// TIA Portal project "project_box_stacking" (V18)
// Vorlageprojekt für das Buch mit Zielsystem S7-1200

(* hardware
DEVICE "S7-1200-Station_1"  S7-1200 Station
   slot 0: "Baugruppenträger_0"  Rack  V1.0
   slot 1: "PLC_1"  CPU 1211C DC/DC/DC  6ES7 211-1AE40-0XB0  V4.1
*)

// ===== PLC "PLC_1"  CPU 1211C DC/DC/DC =====

VAR_GLOBAL   // PLC tag table "Standard-Variablentabelle"
   "FirstScan" AT %M1.0 : Bool;
   "DiagStatusUpdate" AT %M1.1 : Bool;
   "AlwaysTRUE" AT %M1.2 : Bool;
   "AlwaysFALSE" AT %M1.3 : Bool;
   "Clock_Byte" AT %MB0 : Byte;
   "Clock_10Hz" AT %M0.0 : Bool;
   "Clock_5Hz" AT %M0.1 : Bool;
   "Clock_2.5Hz" AT %M0.2 : Bool;
   "Clock_2Hz" AT %M0.3 : Bool;
   "Clock_1.25Hz" AT %M0.4 : Bool;
   "Clock_1Hz" AT %M0.5 : Bool;
   "Clock_0.625Hz" AT %M0.6 : Bool;
   "Clock_0.5Hz" AT %M0.7 : Bool;
   "System_Byte" AT %MB1 : Byte;
END_VAR

VAR_GLOBAL   // PLC tag table " FactoryIO_1"
   "Moving X" AT %I0.0 : Bool;
   "Moving Z" AT %I0.1 : Bool;
   "Item detected" AT %I0.2 : Bool;
   "Lid before place" AT %I0.3 : Bool;
   "Lid clamped" AT %I0.4 : Bool;
   "Pos. at limit (lids)" AT %I0.5 : Bool;
   "Base at place" AT %I0.6 : Bool;
   "Base clamped" AT %I0.7 : Bool;
   "Pos. at limit (bases)" AT %I1.0 : Bool;
   "Part leaving" AT %I1.1 : Bool;
   "Start" AT %I1.2 : Bool;
   "Reset" AT %I1.3 : Bool;
   "Stop" AT %I1.4 : Bool;
   "Emergency stop" AT %I1.5 : Bool;
   "Auto" AT %I1.6 : Bool;
   "FACTORY I/O (Running)" AT %I1.7 : Bool;
   "Grab" AT %Q0.2 : Bool;
   "Lids conveyor" AT %Q0.3 : Bool;
   "Clamp lid" AT %Q0.4 : Bool;
   "Pos. raise (lids)" AT %Q0.5 : Bool;
   "Bases conveyor" AT %Q0.6 : Bool;
   "Pos. raise (bases)" AT %Q1.0 : Bool;
   "Start light" AT %Q1.1 : Bool;
   "Reset light" AT %Q1.2 : Bool;
   "Stop light" AT %Q1.3 : Bool;
   "Counter" AT %QD31 : DInt;
   "Clamp base" AT %Q0.7 : Bool;
   "Move X" AT %Q0.0 : Bool;
   "Move Z" AT %Q0.1 : Bool;
   "Vision sensor Blue lid" AT %I2.4 : Bool;
   "Green Light" AT %Q1.4 : Bool;
   "Counter stacked" AT %I2.3 : Bool;
   "Lid queue" AT %I2.2 : Bool;
   "Sensor stacked" AT %I2.1 : Bool;
   "FACTORY I/O (Reset)" AT %I2.0 : Bool;
   "Vision sensor Blue base" AT %I2.5 : Bool;
   "sensor lid at place" AT %I2.6 : Bool;
   "Base leaving" AT %I2.7 : Bool;
   "Sensor bases at place" AT %I5.3 : Bool;
END_VAR

VAR_GLOBAL   // PLC tag table " FactoryIO_2"
   "Moving X 2" AT %I3.0 : Bool;
   "Moving Z 2" AT %I3.1 : Bool;
   "Item detected 2" AT %I3.2 : Bool;
   "Lid before place 2" AT %I3.3 : Bool;
   "Lid clamped 2" AT %I3.4 : Bool;
   "Pos. at limit (lids) 2" AT %I3.5 : Bool;
   "Base at place 2" AT %I3.6 : Bool;
   "Base clamped 2" AT %I3.7 : Bool;
   "Pos. at limit (bases) 2" AT %I4.0 : Bool;
   "Part leaving 2" AT %I4.1 : Bool;
   "Sensor stacked 2" AT %I4.2 : Bool;
   "Lid queue 2" AT %I4.3 : Bool;
   "Counter stacked 2" AT %I4.4 : Bool;
   "Vision Sensor Green Lid" AT %I4.5 : Bool;
   "Move X 2" AT %Q2.0 : Bool;
   "Move Z 2" AT %Q2.1 : Bool;
   "Grab 2" AT %Q2.2 : Bool;
   "Lids conveyor 2" AT %Q2.3 : Bool;
   "Clamp lid 2" AT %Q2.4 : Bool;
   "Pos. raise (lids) 2" AT %Q2.5 : Bool;
   "Counter 2" AT %QD35 : DInt;
   "Bases conveyor 2" AT %Q2.6 : Bool;
   "Clamp base 2" AT %Q2.7 : Bool;
   "Pos. raise (bases) 2" AT %Q3.0 : Bool;
   "Sensor lid at place 2" AT %I4.6 : Bool;
   "Vision Sensor Green Base" AT %I4.7 : Bool;
   "Base leaving 2" AT %I5.0 : Bool;
   "Sensor base at place 2" AT %I5.1 : Bool;
END_VAR

VAR_GLOBAL   // PLC tag table "markers"
   "m_is_system_on" AT %M3.0 : Bool;
   "m_lid_conveyor" AT %M3.1 : Bool;
   "m_base_conveyor" AT %M3.2 : Bool;
END_VAR

DATA_BLOCK "FB_main_DB"   // DB1
{ S7_Optimized_Access := 'TRUE' }
VERSION : 0.1
// stored: InstanceOfName FB_main
"FB_main"
BEGIN
END_DATA_BLOCK

DATA_BLOCK "FB_main_DB_2"   // DB2
{ S7_Optimized_Access := 'TRUE' }
VERSION : 0.1
// stored: InstanceOfName FB_main
"FB_main"
BEGIN
END_DATA_BLOCK

FUNCTION_BLOCK "FB_main"   // FB1, LAD
{ S7_Optimized_Access := 'TRUE' }
VERSION : 0.1
   VAR_INPUT
      iReset : Bool;   // 'Reset button status' - Observes the reset button, used to reset the system to initial conditions
      iLid_before_place : Bool;   // iLid_at_place - 'Lid presence sensor' - Detects whether a lid is at the required position to be fit
      iItem_detected : Bool;   // 'Item detection sensor' - Identifies the presence of an item in a robotic arm
      iBase_before_place : Bool;   // 'Base presence sensor' - Senses if a base is present at the required position to be fit
      iPart_leaving : Bool;   // Part departure sensor' - Monitors parts leaving a grip area, to control the flow of items.
      iSensor_stacked : Bool;   // 'Stack sensor' - Detects stacked items
      iLid_clamped : Bool;   // - Checks the lid mechanism is clamped,
      iBase_clamped : Bool;   // Checks the basesmechanism is clamped,
      iMoving_Z : Bool;   // Detects movement along the Z-axis,
      iMoving_X : Bool;   // Detects movement along the X-axis
      iLid_queue : Bool;   // Monitors the place before lids grab area
      iCounter_stacked : Bool;   // Stack counter' - Counts the number of stacked items
      iVision_sensor_blue_lid : Bool;   // Blue lid vision sensor' - Vision system input that detects the presence of blue-colored lids;
      iVision_sensor_blue_base : Bool;   // Blue lid vision sensor' - Vision system input that detects the presence of blue-colored lids;
      "iSensor_lid _at_place" : Bool;   // Checks for the presence of a lid at the pick-up point.
      "iSensor_base _at_place" : Bool;   // Checks for the presence of a base at the pick-up point.
      iBase_leaving : Bool;   // "Monitors for a objects leaving pick up point
   END_VAR
   VAR_OUTPUT
      "qLid_ conveyor" : Bool;   // 'Conveyor belt control for lid transport' - Activates the conveyor section responsible for moving lids/parts
      "qBase_ conveyor" : Bool;   // 'Conveyor belt control for base transport' - Activates the conveyor section for moving the base parts
      qClamp_lid : Bool;   // 'Actuate lid clamp' - Engages the mechanism to clamp the lid
      qClamp_base : Bool;   // 'Actuate base clamp' - Engages the mechanism to clamp the base
      qMove_Z : Bool;   // 'Vertical movement actuator' - Controls the vertical movement, likely of a robotic arm
      qMove_X : Bool;   // 'Horizontal movement actuator X-axis' - Controls the horizontal movement along the X-axis
      qGrab : Bool;   // 'Gripping actuator control' - Activates the mechanism to grip an item
      "qPos._raise_lids" : Bool;   // 'Conveyor lids passage control mechanism' - Controls the raising and lowering mechanism
      "qPos._raise_bases" : Bool;   // 'Conveyor bases passage control mechanism' - Controls the raising and lowering mechanism
      qCount_stacked : DInt;   // 'Stack count monitoring' - display the count of stacked items at exit
      qGreen_light : Bool;   // 'Green light indicator' - Activates the green light
   END_VAR
   VAR
      Sequence_lids : Struct
         is_at_place : Bool;
         is_fited : Bool;
         is_grabed : Bool;
         is_above_base : Bool;
      END_STRUCT;
      Sequence_bases : Struct
         at_place : Bool := false;
         is_fited : Bool := false;
      END_STRUCT;
      Sequence_part : Struct
         is_stacked : Bool;
         above_lids_conv : Bool;
         at_place : Bool;
         "exit" : Bool;
      END_STRUCT;
      sequence_no_blue : Struct
         lids : Bool;
         bases : Bool;
      END_STRUCT;
      "array" : Array[0..10] of Bool;
      onemove : Bool;   // System flag to make one operation in program
      Timer_1 : TON_TIME;
      Timer_2 : TON_TIME;
      Timer_3 : TON_TIME;
      Timer_4 : TON_TIME;
      Timer_5 : TON_TIME;
      Timer_6 : TON_TIME;
      Timer_7 : TON_TIME;
      Timer_8 : TON_TIME;
      Timer_9 : TON_TIME;
      Timer_10 : TON_TIME;
      Timer_11 : TON_TIME;
      Timer_12 : TON_TIME;
      "counter" : CTU_INT;   // "stacked parts counter at exit - Tracks the number of completed cycles or parts processed.
   END_VAR
   VAR RETAIN
      reset : Bool;   // System Reset Flag
   END_VAR
   VAR_TEMP   // added for the SCL form of the ladder/FBD networks
      _w1 : Bool;
      _w2 : Bool;
      _w3 : Bool;
   END_VAR
BEGIN

REGION Network 1: init
   // Initialization Routine - Resets control bits and status indicators at system startup or upon reset. Ensures that the system begins operation with a clear configuration
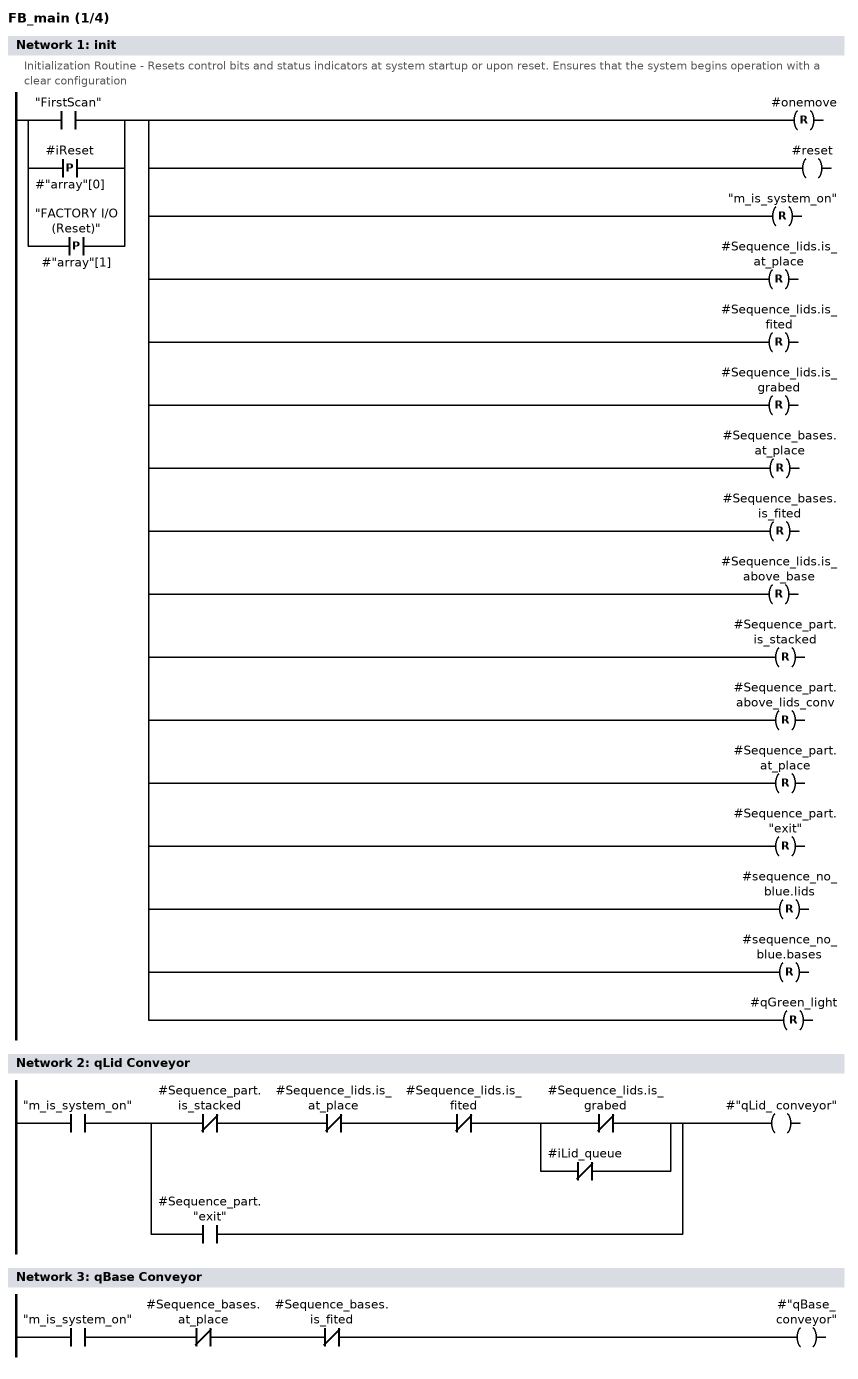
   RUNG wire#powerrail
      Contact( "FirstScan" )
      wire#w1
      R_Coil( #onemove )
   END_RUNG
   RUNG wire#powerrail
      P_Contact(operand := #iReset, bit := #"array"[0])
   END_RUNG wire#w1
   RUNG wire#powerrail
      P_Contact(operand := "FACTORY I/O (Reset)", bit := #"array"[1])
   END_RUNG wire#w1
   RUNG wire#w1
      Coil( #reset )
   END_RUNG
   RUNG wire#w1
      R_Coil( "m_is_system_on" )
   END_RUNG
   RUNG wire#w1
      R_Coil( #Sequence_lids.is_at_place )
   END_RUNG
   RUNG wire#w1
      R_Coil( #Sequence_lids.is_fited )
   END_RUNG
   RUNG wire#w1
      R_Coil( #Sequence_lids.is_grabed )
   END_RUNG
   RUNG wire#w1
      R_Coil( #Sequence_bases.at_place )
   END_RUNG
   RUNG wire#w1
      R_Coil( #Sequence_bases.is_fited )
   END_RUNG
   RUNG wire#w1
      R_Coil( #Sequence_lids.is_above_base )
   END_RUNG
   RUNG wire#w1
      R_Coil( #Sequence_part.is_stacked )
   END_RUNG
   RUNG wire#w1
      R_Coil( #Sequence_part.above_lids_conv )
   END_RUNG
   RUNG wire#w1
      R_Coil( #Sequence_part.at_place )
   END_RUNG
   RUNG wire#w1
      R_Coil( #Sequence_part."exit" )
   END_RUNG
   RUNG wire#w1
      R_Coil( #sequence_no_blue.lids )
   END_RUNG
   RUNG wire#w1
      R_Coil( #sequence_no_blue.bases )
   END_RUNG
   RUNG wire#w1
      R_Coil( #qGreen_light )
   END_RUNG
   // the same network as SCL:
   #_w1 := #iReset AND NOT #"array"[0];   // rising edge of #iReset
   #"array"[0] := #iReset;
   #_w2 := "FACTORY I/O (Reset)" AND NOT #"array"[1];   // rising edge of "FACTORY I/O (Reset)"
   #"array"[1] := "FACTORY I/O (Reset)";
   #_w3 := "FirstScan" OR #_w1 OR #_w2;
   IF #_w3 THEN #onemove := FALSE; END_IF;
   #reset := #_w3;
   IF #_w3 THEN
       "m_is_system_on" := FALSE;
       #Sequence_lids.is_at_place := FALSE;
       #Sequence_lids.is_fited := FALSE;
       #Sequence_lids.is_grabed := FALSE;
       #Sequence_bases.at_place := FALSE;
       #Sequence_bases.is_fited := FALSE;
       #Sequence_lids.is_above_base := FALSE;
       #Sequence_part.is_stacked := FALSE;
       #Sequence_part.above_lids_conv := FALSE;
       #Sequence_part.at_place := FALSE;
       #Sequence_part."exit" := FALSE;
       #sequence_no_blue.lids := FALSE;
       #sequence_no_blue.bases := FALSE;
       #qGreen_light := FALSE;
   END_IF;
END_REGION

REGION Network 2: qLid Conveyor
   RUNG wire#powerrail
      Contact( "m_is_system_on" )
      wire#w1
      I_Contact( #Sequence_part.is_stacked )
      I_Contact( #Sequence_lids.is_at_place )
      I_Contact( #Sequence_lids.is_fited )
      wire#w2
      I_Contact( #Sequence_lids.is_grabed )
      wire#w3
      Coil( #"qLid_ conveyor" )
   END_RUNG
   RUNG wire#w2
      I_Contact( #iLid_queue )
   END_RUNG wire#w3
   RUNG wire#w1
      Contact( #Sequence_part."exit" )
   END_RUNG wire#w3
   // the same network as SCL:
   #"qLid_ conveyor" := "m_is_system_on" AND ((NOT #Sequence_part.is_stacked AND NOT #Sequence_lids.is_at_place AND NOT #Sequence_lids.is_fited AND (NOT #Sequence_lids.is_grabed OR NOT #iLid_queue)) OR #Sequence_part."exit");
END_REGION

REGION Network 3: qBase Conveyor
   RUNG wire#powerrail
      Contact( "m_is_system_on" )
      I_Contact( #Sequence_bases.at_place )
      I_Contact( #Sequence_bases.is_fited )
      Coil( #"qBase_ conveyor" )
   END_RUNG
   // the same network as SCL:
   #"qBase_ conveyor" := "m_is_system_on" AND NOT #Sequence_bases.at_place AND NOT #Sequence_bases.is_fited;
END_REGION

REGION Network 4: qClamp lid
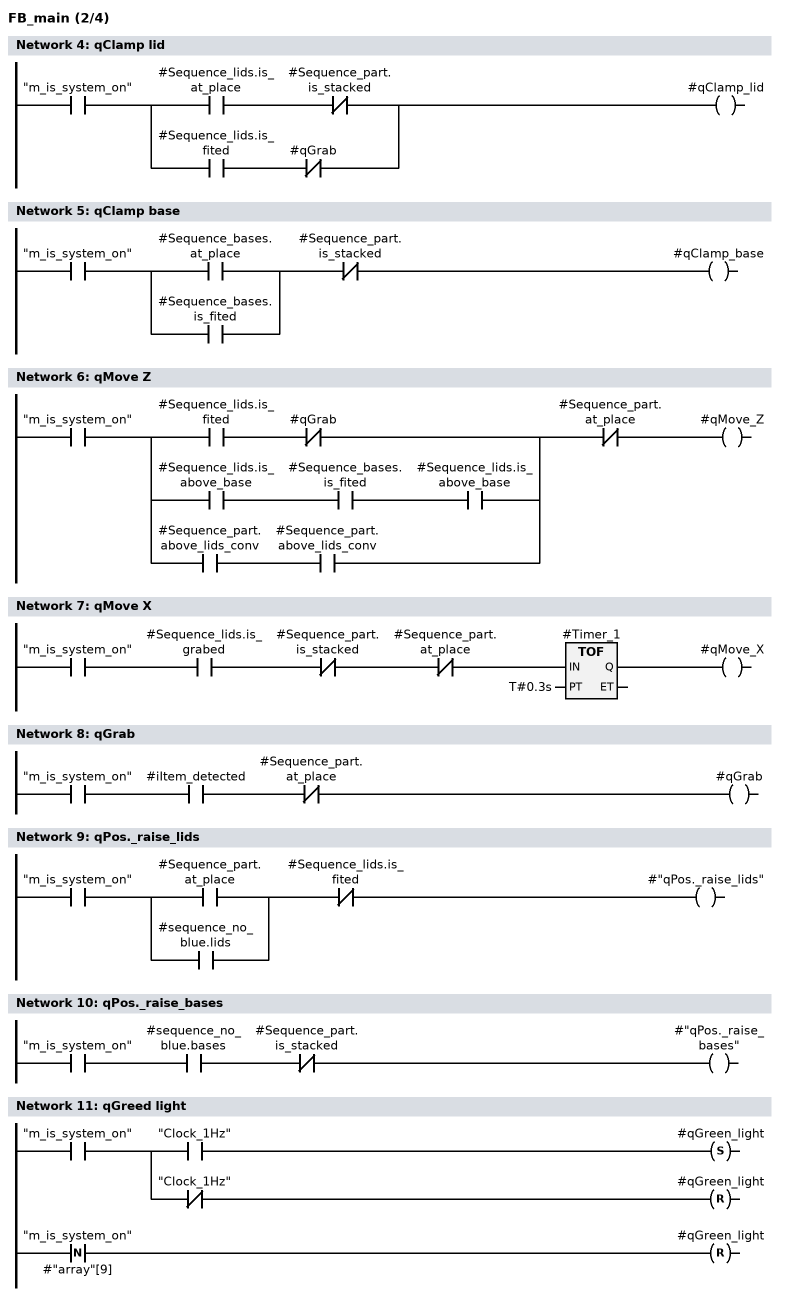
   RUNG wire#powerrail
      Contact( "m_is_system_on" )
      wire#w1
      Contact( #Sequence_lids.is_at_place )
      I_Contact( #Sequence_part.is_stacked )
      wire#w2
      Coil( #qClamp_lid )
   END_RUNG
   RUNG wire#w1
      Contact( #Sequence_lids.is_fited )
      I_Contact( #qGrab )
   END_RUNG wire#w2
   // the same network as SCL:
   #qClamp_lid := "m_is_system_on" AND ((#Sequence_lids.is_at_place AND NOT #Sequence_part.is_stacked) OR (#Sequence_lids.is_fited AND NOT #qGrab));
END_REGION

REGION Network 5: qClamp base
   RUNG wire#powerrail
      Contact( "m_is_system_on" )
      wire#w1
      Contact( #Sequence_bases.at_place )
      wire#w2
      I_Contact( #Sequence_part.is_stacked )
      Coil( #qClamp_base )
   END_RUNG
   RUNG wire#w1
      Contact( #Sequence_bases.is_fited )
   END_RUNG wire#w2
   // the same network as SCL:
   #qClamp_base := "m_is_system_on" AND (#Sequence_bases.at_place OR #Sequence_bases.is_fited) AND NOT #Sequence_part.is_stacked;
END_REGION

REGION Network 6: qMove Z
   RUNG wire#powerrail
      Contact( "m_is_system_on" )
      wire#w1
      Contact( #Sequence_lids.is_fited )
      I_Contact( #qGrab )
      wire#w2
      I_Contact( #Sequence_part.at_place )
      Coil( #qMove_Z )
   END_RUNG
   RUNG wire#w1
      Contact( #Sequence_lids.is_above_base )
      Contact( #Sequence_bases.is_fited )
      Contact( #Sequence_lids.is_above_base )
   END_RUNG wire#w2
   RUNG wire#w1
      Contact( #Sequence_part.above_lids_conv )
      Contact( #Sequence_part.above_lids_conv )
   END_RUNG wire#w2
   // the same network as SCL:
   #qMove_Z := "m_is_system_on" AND ((#Sequence_lids.is_fited AND NOT #qGrab) OR (#Sequence_lids.is_above_base AND #Sequence_bases.is_fited AND #Sequence_lids.is_above_base) OR (#Sequence_part.above_lids_conv AND #Sequence_part.above_lids_conv)) AND NOT #Sequence_part.at_place;
END_REGION

REGION Network 7: qMove X
   #Timer_1(IN := "m_is_system_on" AND #Sequence_lids.is_grabed AND NOT #Sequence_part.is_stacked AND NOT #Sequence_part.at_place,   // TOF
            PT := T#0.3s);
   #qMove_X := #Timer_1.Q;
END_REGION

REGION Network 8: qGrab
   RUNG wire#powerrail
      Contact( "m_is_system_on" )
      Contact( #iItem_detected )
      I_Contact( #Sequence_part.at_place )
      Coil( #qGrab )
   END_RUNG
   // the same network as SCL:
   #qGrab := "m_is_system_on" AND #iItem_detected AND NOT #Sequence_part.at_place;
END_REGION

REGION Network 9: qPos._raise_lids
   RUNG wire#powerrail
      Contact( "m_is_system_on" )
      wire#w1
      Contact( #Sequence_part.at_place )
      wire#w2
      I_Contact( #Sequence_lids.is_fited )
      Coil( #"qPos._raise_lids" )
   END_RUNG
   RUNG wire#w1
      Contact( #sequence_no_blue.lids )
   END_RUNG wire#w2
   // the same network as SCL:
   #"qPos._raise_lids" := "m_is_system_on" AND (#Sequence_part.at_place OR #sequence_no_blue.lids) AND NOT #Sequence_lids.is_fited;
END_REGION

REGION Network 10: qPos._raise_bases
   RUNG wire#powerrail
      Contact( "m_is_system_on" )
      Contact( #sequence_no_blue.bases )
      I_Contact( #Sequence_part.is_stacked )
      Coil( #"qPos._raise_bases" )
   END_RUNG
   // the same network as SCL:
   #"qPos._raise_bases" := "m_is_system_on" AND #sequence_no_blue.bases AND NOT #Sequence_part.is_stacked;
END_REGION

REGION Network 11: qGreed light
   RUNG wire#powerrail
      Contact( "m_is_system_on" )
      wire#w1
      Contact( "Clock_1Hz" )
      S_Coil( #qGreen_light )
   END_RUNG
   RUNG wire#w1
      I_Contact( "Clock_1Hz" )
      R_Coil( #qGreen_light )
   END_RUNG
   RUNG wire#powerrail
      N_Contact(operand := "m_is_system_on", bit := #"array"[9])
      R_Coil( #qGreen_light )
   END_RUNG
   // the same network as SCL:
   IF "m_is_system_on" AND "Clock_1Hz" THEN #qGreen_light := TRUE; END_IF;
   IF "m_is_system_on" AND NOT "Clock_1Hz" THEN #qGreen_light := FALSE; END_IF;
   #_w1 := NOT "m_is_system_on" AND #"array"[9];   // falling edge of "m_is_system_on"
   #"array"[9] := "m_is_system_on";
   IF #_w1 THEN #qGreen_light := FALSE; END_IF;
END_REGION

REGION Network 12: Sequence lids at place
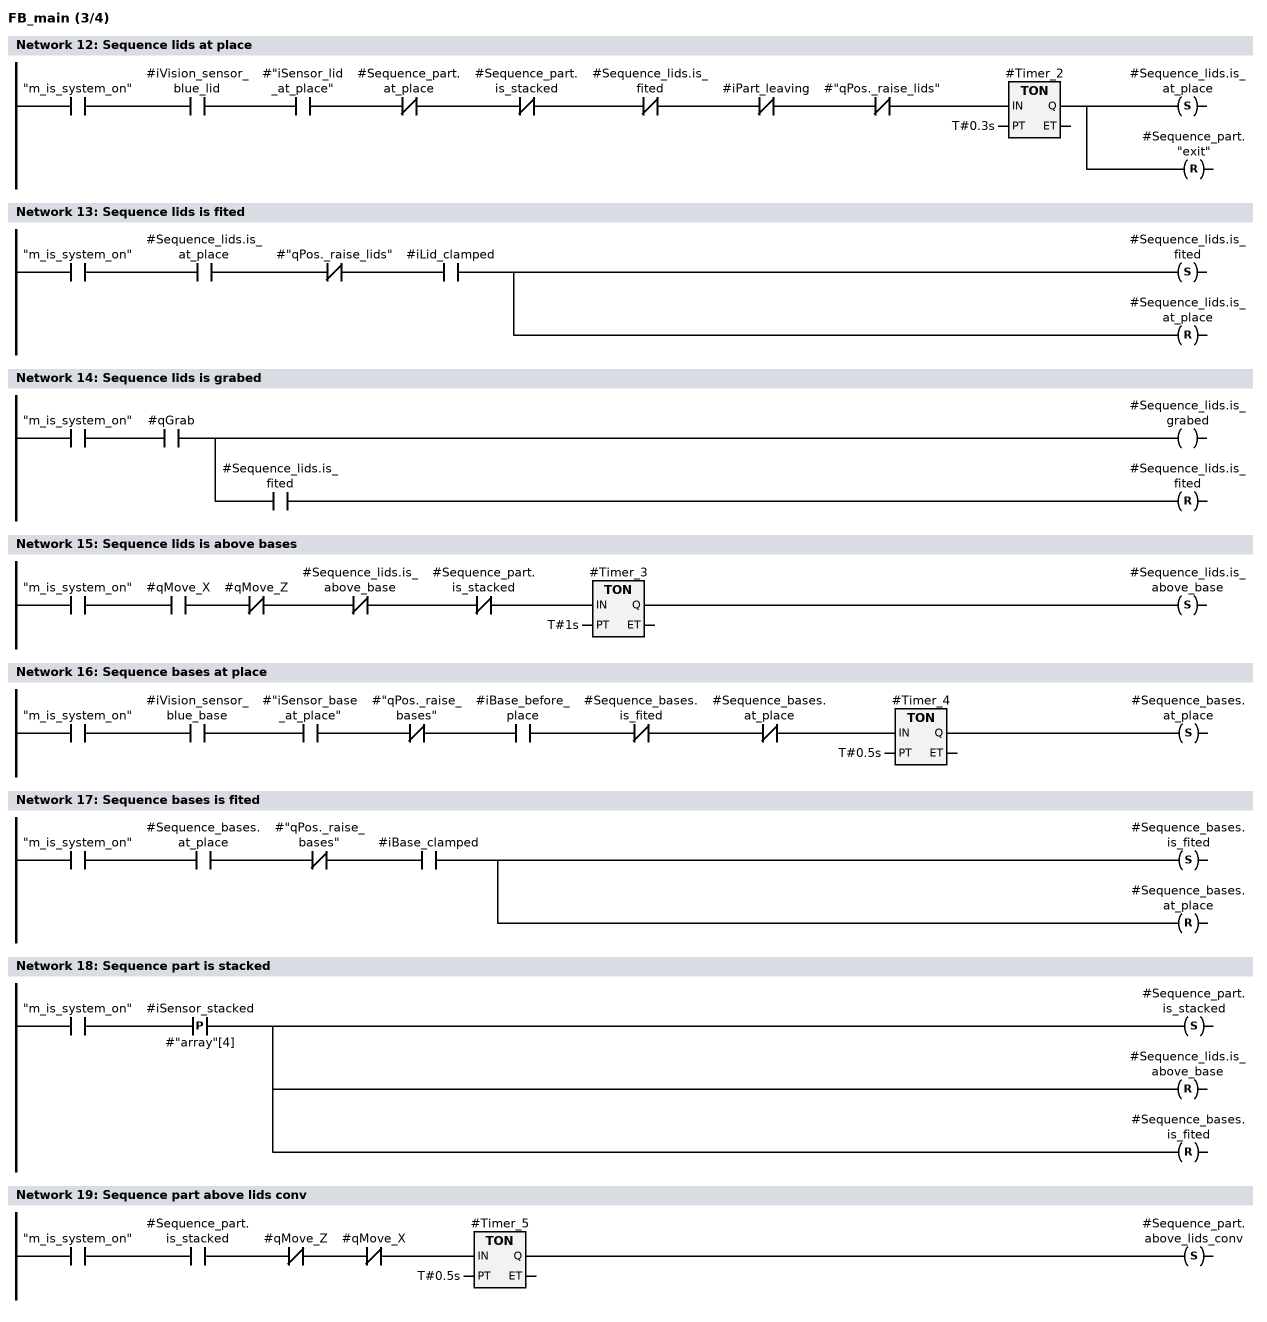
   #Timer_2(IN := "m_is_system_on" AND #iVision_sensor_blue_lid AND #"iSensor_lid _at_place" AND NOT #Sequence_part.at_place AND NOT #Sequence_part.is_stacked AND NOT #Sequence_lids.is_fited AND NOT #iPart_leaving AND NOT #"qPos._raise_lids",   // TON
            PT := T#0.3s);
   IF #Timer_2.Q THEN
       #Sequence_lids.is_at_place := TRUE;
       #Sequence_part."exit" := FALSE;
   END_IF;
END_REGION

REGION Network 13: Sequence lids is fited
   RUNG wire#powerrail
      Contact( "m_is_system_on" )
      Contact( #Sequence_lids.is_at_place )
      I_Contact( #"qPos._raise_lids" )
      Contact( #iLid_clamped )
      wire#w1
      S_Coil( #Sequence_lids.is_fited )
   END_RUNG
   RUNG wire#w1
      R_Coil( #Sequence_lids.is_at_place )
   END_RUNG
   // the same network as SCL:
   IF "m_is_system_on" AND #Sequence_lids.is_at_place AND NOT #"qPos._raise_lids" AND #iLid_clamped THEN
       #Sequence_lids.is_fited := TRUE;
       #Sequence_lids.is_at_place := FALSE;
   END_IF;
END_REGION

REGION Network 14: Sequence lids is grabed
   RUNG wire#powerrail
      Contact( "m_is_system_on" )
      Contact( #qGrab )
      wire#w1
      Coil( #Sequence_lids.is_grabed )
   END_RUNG
   RUNG wire#w1
      Contact( #Sequence_lids.is_fited )
      R_Coil( #Sequence_lids.is_fited )
   END_RUNG
   // the same network as SCL:
   #Sequence_lids.is_grabed := "m_is_system_on" AND #qGrab;
   IF #Sequence_lids.is_grabed AND #Sequence_lids.is_fited THEN #Sequence_lids.is_fited := FALSE; END_IF;
END_REGION

REGION Network 15: Sequence lids is above bases
   #Timer_3(IN := "m_is_system_on" AND #qMove_X AND NOT #qMove_Z AND NOT #Sequence_lids.is_above_base AND NOT #Sequence_part.is_stacked,   // TON
            PT := T#1s);
   IF #Timer_3.Q THEN #Sequence_lids.is_above_base := TRUE; END_IF;
END_REGION

REGION Network 16: Sequence bases at place
   #Timer_4(IN := "m_is_system_on" AND #iVision_sensor_blue_base AND #"iSensor_base _at_place" AND NOT #"qPos._raise_bases" AND #iBase_before_place AND NOT #Sequence_bases.is_fited AND NOT #Sequence_bases.at_place,   // TON
            PT := T#0.5s);
   IF #Timer_4.Q THEN #Sequence_bases.at_place := TRUE; END_IF;
END_REGION

REGION Network 17: Sequence bases is fited
   RUNG wire#powerrail
      Contact( "m_is_system_on" )
      Contact( #Sequence_bases.at_place )
      I_Contact( #"qPos._raise_bases" )
      Contact( #iBase_clamped )
      wire#w1
      S_Coil( #Sequence_bases.is_fited )
   END_RUNG
   RUNG wire#w1
      R_Coil( #Sequence_bases.at_place )
   END_RUNG
   // the same network as SCL:
   IF "m_is_system_on" AND #Sequence_bases.at_place AND NOT #"qPos._raise_bases" AND #iBase_clamped THEN
       #Sequence_bases.is_fited := TRUE;
       #Sequence_bases.at_place := FALSE;
   END_IF;
END_REGION

REGION Network 18: Sequence part is stacked
   RUNG wire#powerrail
      Contact( "m_is_system_on" )
      P_Contact(operand := #iSensor_stacked, bit := #"array"[4])
      wire#w1
      S_Coil( #Sequence_part.is_stacked )
   END_RUNG
   RUNG wire#w1
      R_Coil( #Sequence_lids.is_above_base )
   END_RUNG
   RUNG wire#w1
      R_Coil( #Sequence_bases.is_fited )
   END_RUNG
   // the same network as SCL:
   #_w1 := "m_is_system_on" AND #iSensor_stacked AND NOT #"array"[4];   // rising edge of #iSensor_stacked
   #"array"[4] := #iSensor_stacked;
   IF #_w1 THEN
       #Sequence_part.is_stacked := TRUE;
       #Sequence_lids.is_above_base := FALSE;
       #Sequence_bases.is_fited := FALSE;
   END_IF;
END_REGION

REGION Network 19: Sequence part above lids conv
   #Timer_5(IN := "m_is_system_on" AND #Sequence_part.is_stacked AND NOT #qMove_Z AND NOT #qMove_X,   // TON
            PT := T#0.5s);
   IF #Timer_5.Q THEN #Sequence_part.above_lids_conv := TRUE; END_IF;
END_REGION

REGION Network 20: Sequence part at place
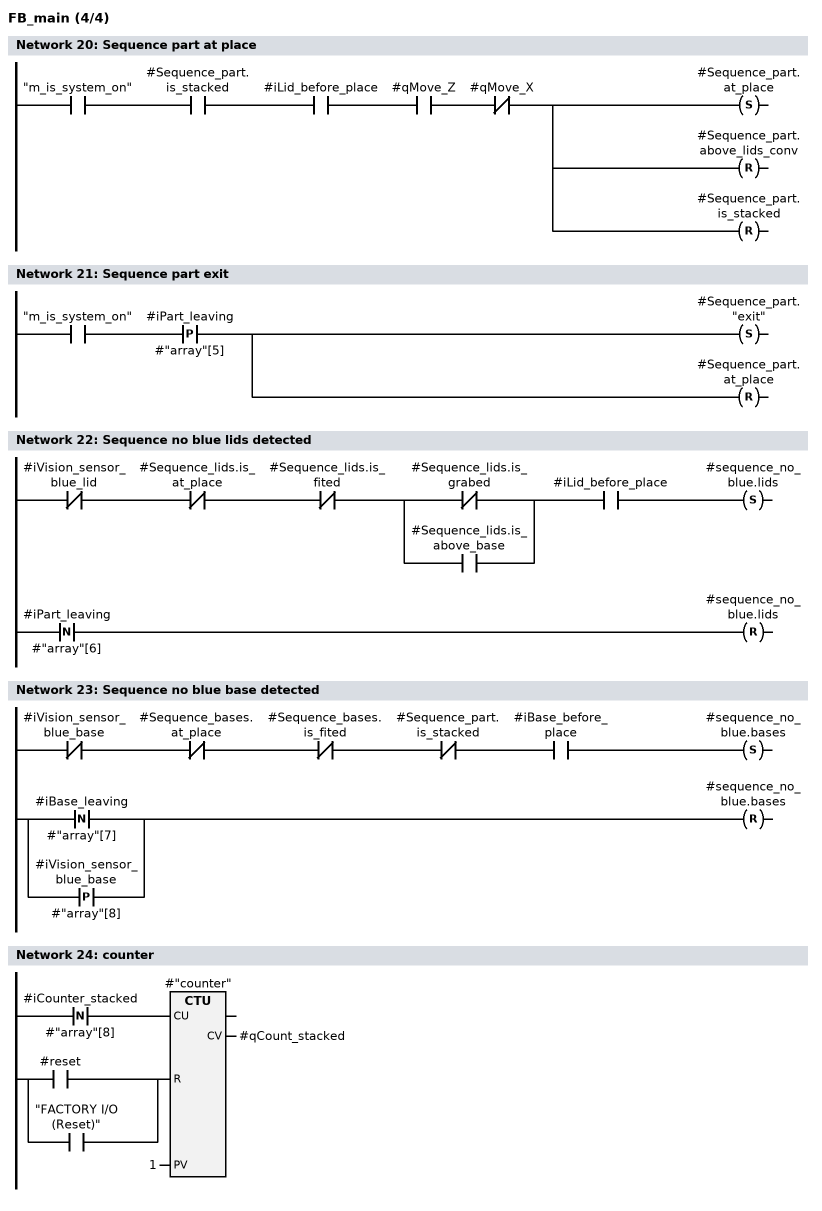
   RUNG wire#powerrail
      Contact( "m_is_system_on" )
      Contact( #Sequence_part.is_stacked )
      Contact( #iLid_before_place )
      Contact( #qMove_Z )
      I_Contact( #qMove_X )
      wire#w1
      S_Coil( #Sequence_part.at_place )
   END_RUNG
   RUNG wire#w1
      R_Coil( #Sequence_part.above_lids_conv )
   END_RUNG
   RUNG wire#w1
      R_Coil( #Sequence_part.is_stacked )
   END_RUNG
   // the same network as SCL:
   IF "m_is_system_on" AND #Sequence_part.is_stacked AND #iLid_before_place AND #qMove_Z AND NOT #qMove_X THEN
       #Sequence_part.at_place := TRUE;
       #Sequence_part.above_lids_conv := FALSE;
       #Sequence_part.is_stacked := FALSE;
   END_IF;
END_REGION

REGION Network 21: Sequence part exit
   RUNG wire#powerrail
      Contact( "m_is_system_on" )
      P_Contact(operand := #iPart_leaving, bit := #"array"[5])
      wire#w1
      S_Coil( #Sequence_part."exit" )
   END_RUNG
   RUNG wire#w1
      R_Coil( #Sequence_part.at_place )
   END_RUNG
   // the same network as SCL:
   #_w1 := "m_is_system_on" AND #iPart_leaving AND NOT #"array"[5];   // rising edge of #iPart_leaving
   #"array"[5] := #iPart_leaving;
   IF #_w1 THEN
       #Sequence_part."exit" := TRUE;
       #Sequence_part.at_place := FALSE;
   END_IF;
END_REGION

REGION Network 22: Sequence no blue lids detected
   RUNG wire#powerrail
      I_Contact( #iVision_sensor_blue_lid )
      I_Contact( #Sequence_lids.is_at_place )
      I_Contact( #Sequence_lids.is_fited )
      wire#w1
      I_Contact( #Sequence_lids.is_grabed )
      wire#w2
      Contact( #iLid_before_place )
      S_Coil( #sequence_no_blue.lids )
   END_RUNG
   RUNG wire#w1
      Contact( #Sequence_lids.is_above_base )
   END_RUNG wire#w2
   RUNG wire#powerrail
      N_Contact(operand := #iPart_leaving, bit := #"array"[6])
      R_Coil( #sequence_no_blue.lids )
   END_RUNG
   // the same network as SCL:
   IF NOT #iVision_sensor_blue_lid AND NOT #Sequence_lids.is_at_place AND NOT #Sequence_lids.is_fited AND (NOT #Sequence_lids.is_grabed OR #Sequence_lids.is_above_base) AND #iLid_before_place THEN
       #sequence_no_blue.lids := TRUE;
   END_IF;
   #_w1 := NOT #iPart_leaving AND #"array"[6];   // falling edge of #iPart_leaving
   #"array"[6] := #iPart_leaving;
   IF #_w1 THEN #sequence_no_blue.lids := FALSE; END_IF;
END_REGION

REGION Network 23: Sequence no blue base detected
   RUNG wire#powerrail
      I_Contact( #iVision_sensor_blue_base )
      I_Contact( #Sequence_bases.at_place )
      I_Contact( #Sequence_bases.is_fited )
      I_Contact( #Sequence_part.is_stacked )
      Contact( #iBase_before_place )
      S_Coil( #sequence_no_blue.bases )
   END_RUNG
   RUNG wire#powerrail
      N_Contact(operand := #iBase_leaving, bit := #"array"[7])
      wire#w1
      R_Coil( #sequence_no_blue.bases )
   END_RUNG
   RUNG wire#powerrail
      P_Contact(operand := #iVision_sensor_blue_base, bit := #"array"[8])
   END_RUNG wire#w1
   // the same network as SCL:
   IF NOT #iVision_sensor_blue_base AND NOT #Sequence_bases.at_place AND NOT #Sequence_bases.is_fited AND NOT #Sequence_part.is_stacked AND #iBase_before_place THEN
       #sequence_no_blue.bases := TRUE;
   END_IF;
   #_w1 := NOT #iBase_leaving AND #"array"[7];   // falling edge of #iBase_leaving
   #"array"[7] := #iBase_leaving;
   #_w2 := #iVision_sensor_blue_base AND NOT #"array"[8];   // rising edge of #iVision_sensor_blue_base
   #"array"[8] := #iVision_sensor_blue_base;
   IF #_w1 OR #_w2 THEN #sequence_no_blue.bases := FALSE; END_IF;
END_REGION

REGION Network 24: counter
   #_w1 := NOT #iCounter_stacked AND #"array"[8];   // falling edge of #iCounter_stacked
   #"array"[8] := #iCounter_stacked;
   #"counter"(CU := #_w1, R := #reset OR "FACTORY I/O (Reset)", PV := 1, CV => #qCount_stacked);   // CTU
END_REGION

REGION Network 25: need to base conveyor
END_REGION
END_FUNCTION_BLOCK

FUNCTION "system on/off" : Void   // FC1, LAD
{ S7_Optimized_Access := 'TRUE' }
VERSION : 0.1
   VAR_INPUT
      iStart_button : Bool;
      iStop_button : Bool;
   END_VAR
BEGIN

REGION Network 1
   // System Control Logic - Monitors the start and stop conditions to maintain the system's operational state. Ensures that the system can only be started if it is not signaled to stop or reset.
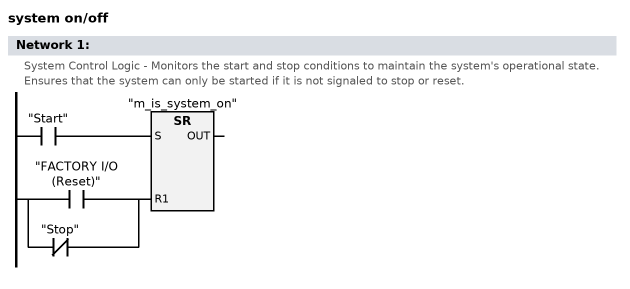
   RUNG wire#powerrail
      Contact( "Start" )
      S_SR(operand := "m_is_system_on", r1 := wire#w1)
   END_RUNG
   RUNG wire#powerrail
      Contact( "FACTORY I/O (Reset)" )
   END_RUNG wire#w1
   RUNG wire#powerrail
      I_Contact( "Stop" )
   END_RUNG wire#w1
   // the same network as SCL:
   IF "Start" THEN
       "m_is_system_on" := TRUE;   // SR flip-flop
   END_IF;
   IF "FACTORY I/O (Reset)" OR NOT "Stop" THEN "m_is_system_on" := FALSE; END_IF;
END_REGION
END_FUNCTION

FUNCTION "MHJ-PLC-Lab-Function-S71200" : Void   // FC9000, SCL
{ S7_Optimized_Access := 'TRUE' }
VERSION : 0.1
   VAR_TEMP
      rdTimeReturn : Int;
      outputTime : DTL;
      SyncVal : Byte;
      forVal : Int;
      forVal_2 : Int;
      Value : Byte;
   END_VAR
   VAR CONSTANT
      CompVal : Byte := 16#34;
      Value_01 : Byte := 16#11;
      Value_01_DW : DWord := 16#A165_D992;
      Value_02_DW : DWord := 16#58BE_4401;
   END_VAR
BEGIN

   #Value:=PEEK(area := 16#82,
        dbNumber := 0,
        byteOffset := 511);
   #Value := #Value + 1;

   POKE(area := 16#82,
        dbNumber := 0,
        byteOffset := 511,
        value := #Value);

   POKE(area:=16#81,
        dbNumber:=0,
        byteOffset:=1016,
        value:=#Value_01_DW);
   POKE(area := 16#81,
        dbNumber := 0,
        byteOffset := 1020,
        value := #Value_02_DW);

   POKE(area := 16#81,
        dbNumber := 0,
        byteOffset := 511,
        value := B#16#00);

   FOR #forVal := 0 TO 120 DO
       FOR #forVal_2:=0 TO 10 DO
           #rdTimeReturn:=RD_SYS_T(#outputTime);
           #rdTimeReturn := WR_SYS_T(#outputTime);
           #rdTimeReturn := RD_SYS_T(#outputTime);
           #rdTimeReturn := WR_SYS_T(#outputTime);
       END_FOR;
       #SyncVal:= PEEK(area := 16#81,
                      dbNumber := 0,
                      byteOffset := 511);
       IF #SyncVal = #CompVal THEN
          GOTO M_1;
       END_IF;
   END_FOR;
   RETURN;

   M_1:
   POKE(area := 16#81,
        dbNumber := 0,
        byteOffset := 511,
        value := B#16#0);
END_FUNCTION

ORGANIZATION_BLOCK "Main"   // OB1, LAD, ProgramCycle
TITLE = "Main Program Sweep (Cycle)"
{ S7_Optimized_Access := 'TRUE' }
VERSION : 0.1
   VAR_INPUT
      Initial_Call : Bool;   // Initial call of this OB
      Remanence : Bool;   // =True, if remanent data are available
   END_VAR
BEGIN

REGION Network 1: Konnektierungsbaustein für PLC-Lab
   // Im Netzwerk 1 wird der Konnektierungsbaustein für PLC-Lab aufgerufen.
   // Dieser Aufruf darf nicht entfernt werden!
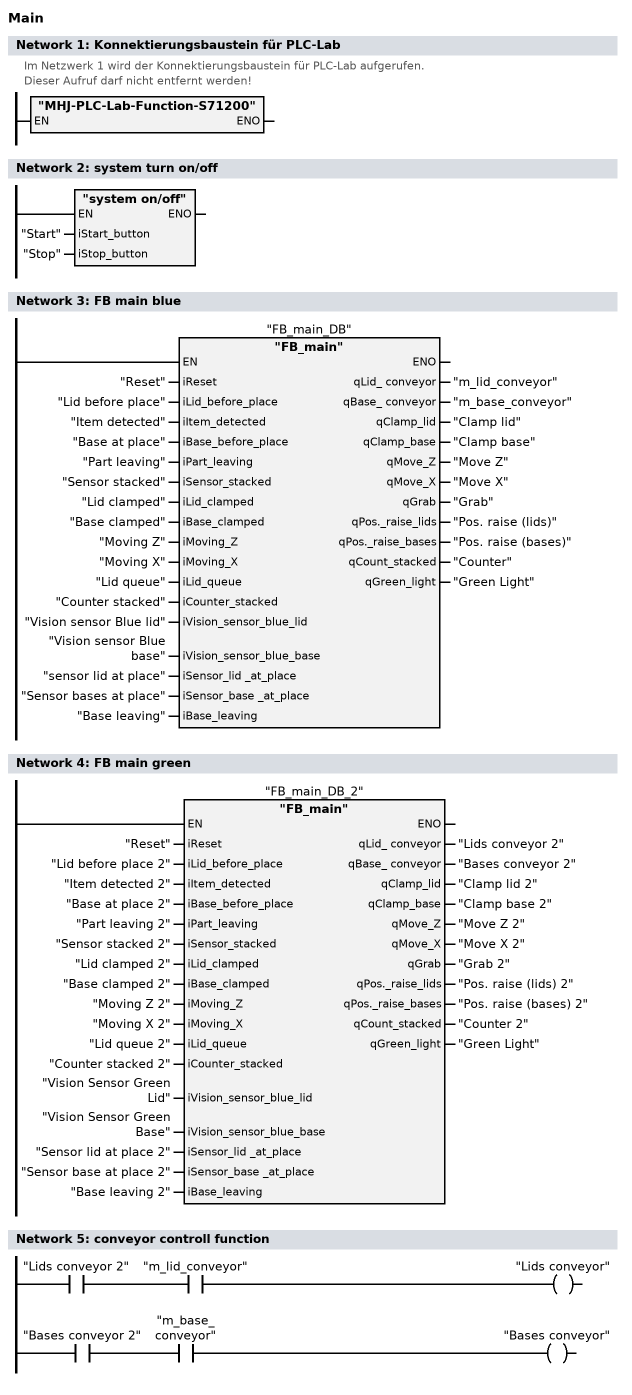
   RUNG wire#powerrail
      "MHJ-PLC-Lab-Function-S71200"()
   END_RUNG
   // the same network as SCL:
   "MHJ-PLC-Lab-Function-S71200"();
END_REGION

REGION Network 2: system turn on/off
   RUNG wire#powerrail
      "system on/off"(iStart_button := "Start", iStop_button := "Stop")
   END_RUNG
   // the same network as SCL:
   "system on/off"(iStart_button := "Start", iStop_button := "Stop");
END_REGION

REGION Network 3: FB main blue
   RUNG wire#powerrail
      "FB_main_DB"(iReset := "Reset", iLid_before_place := "Lid before place", iItem_detected := "Item detected", iBase_before_place := "Base at place", iPart_leaving := "Part leaving", iSensor_stacked := "Sensor stacked", iLid_clamped := "Lid clamped", iBase_clamped := "Base clamped", iMoving_Z := "Moving Z", iMoving_X := "Moving X", iLid_queue := "Lid queue", iCounter_stacked := "Counter stacked", iVision_sensor_blue_lid := "Vision sensor Blue lid", iVision_sensor_blue_base := "Vision sensor Blue base", "iSensor_lid _at_place" := "sensor lid at place", "iSensor_base _at_place" := "Sensor bases at place", iBase_leaving := "Base leaving", "qLid_ conveyor" => "m_lid_conveyor", "qBase_ conveyor" => "m_base_conveyor", qClamp_lid => "Clamp lid", qClamp_base => "Clamp base", qMove_Z => "Move Z", qMove_X => "Move X", qGrab => "Grab", "qPos._raise_lids" => "Pos. raise (lids)", "qPos._raise_bases" => "Pos. raise (bases)", qCount_stacked => "Counter", qGreen_light => "Green Light")
   END_RUNG
   // the same network as SCL:
   "FB_main_DB"(iReset := "Reset",   // "FB_main"
                iLid_before_place := "Lid before place",
                iItem_detected := "Item detected",
                iBase_before_place := "Base at place",
                iPart_leaving := "Part leaving",
                iSensor_stacked := "Sensor stacked",
                iLid_clamped := "Lid clamped",
                iBase_clamped := "Base clamped",
                iMoving_Z := "Moving Z",
                iMoving_X := "Moving X",
                iLid_queue := "Lid queue",
                iCounter_stacked := "Counter stacked",
                iVision_sensor_blue_lid := "Vision sensor Blue lid",
                iVision_sensor_blue_base := "Vision sensor Blue base",
                "iSensor_lid _at_place" := "sensor lid at place",
                "iSensor_base _at_place" := "Sensor bases at place",
                iBase_leaving := "Base leaving",
                "qLid_ conveyor" => "m_lid_conveyor",
                "qBase_ conveyor" => "m_base_conveyor",
                qClamp_lid => "Clamp lid",
                qClamp_base => "Clamp base",
                qMove_Z => "Move Z",
                qMove_X => "Move X",
                qGrab => "Grab",
                "qPos._raise_lids" => "Pos. raise (lids)",
                "qPos._raise_bases" => "Pos. raise (bases)",
                qCount_stacked => "Counter",
                qGreen_light => "Green Light");
END_REGION

REGION Network 4: FB main green
   RUNG wire#powerrail
      "FB_main_DB_2"(iReset := "Reset", iLid_before_place := "Lid before place 2", iItem_detected := "Item detected 2", iBase_before_place := "Base at place 2", iPart_leaving := "Part leaving 2", iSensor_stacked := "Sensor stacked 2", iLid_clamped := "Lid clamped 2", iBase_clamped := "Base clamped 2", iMoving_Z := "Moving Z 2", iMoving_X := "Moving X 2", iLid_queue := "Lid queue 2", iCounter_stacked := "Counter stacked 2", iVision_sensor_blue_lid := "Vision Sensor Green Lid", iVision_sensor_blue_base := "Vision Sensor Green Base", "iSensor_lid _at_place" := "Sensor lid at place 2", "iSensor_base _at_place" := "Sensor base at place 2", iBase_leaving := "Base leaving 2", "qLid_ conveyor" => "Lids conveyor 2", "qBase_ conveyor" => "Bases conveyor 2", qClamp_lid => "Clamp lid 2", qClamp_base => "Clamp base 2", qMove_Z => "Move Z 2", qMove_X => "Move X 2", qGrab => "Grab 2", "qPos._raise_lids" => "Pos. raise (lids) 2", "qPos._raise_bases" => "Pos. raise (bases) 2", qCount_stacked => "Counter 2", qGreen_light => "Green Light")
   END_RUNG
   // the same network as SCL:
   "FB_main_DB_2"(iReset := "Reset",   // "FB_main"
                  iLid_before_place := "Lid before place 2",
                  iItem_detected := "Item detected 2",
                  iBase_before_place := "Base at place 2",
                  iPart_leaving := "Part leaving 2",
                  iSensor_stacked := "Sensor stacked 2",
                  iLid_clamped := "Lid clamped 2",
                  iBase_clamped := "Base clamped 2",
                  iMoving_Z := "Moving Z 2",
                  iMoving_X := "Moving X 2",
                  iLid_queue := "Lid queue 2",
                  iCounter_stacked := "Counter stacked 2",
                  iVision_sensor_blue_lid := "Vision Sensor Green Lid",
                  iVision_sensor_blue_base := "Vision Sensor Green Base",
                  "iSensor_lid _at_place" := "Sensor lid at place 2",
                  "iSensor_base _at_place" := "Sensor base at place 2",
                  iBase_leaving := "Base leaving 2",
                  "qLid_ conveyor" => "Lids conveyor 2",
                  "qBase_ conveyor" => "Bases conveyor 2",
                  qClamp_lid => "Clamp lid 2",
                  qClamp_base => "Clamp base 2",
                  qMove_Z => "Move Z 2",
                  qMove_X => "Move X 2",
                  qGrab => "Grab 2",
                  "qPos._raise_lids" => "Pos. raise (lids) 2",
                  "qPos._raise_bases" => "Pos. raise (bases) 2",
                  qCount_stacked => "Counter 2",
                  qGreen_light => "Green Light");
END_REGION

REGION Network 5: conveyor controll function
   RUNG wire#powerrail
      Contact( "Lids conveyor 2" )
      Contact( "m_lid_conveyor" )
      Coil( "Lids conveyor" )
   END_RUNG
   RUNG wire#powerrail
      Contact( "Bases conveyor 2" )
      Contact( "m_base_conveyor" )
      Coil( "Bases conveyor" )
   END_RUNG
   // the same network as SCL:
   "Lids conveyor" := "Lids conveyor 2" AND "m_lid_conveyor";
   "Bases conveyor" := "Bases conveyor 2" AND "m_base_conveyor";
END_REGION
END_ORGANIZATION_BLOCK